TYPE ST_AxisError:
STRUCT
//PLCopen function block errors
    nPowerErrorID: UDINT; //Error ID MC_Power function block
    nMoveAbsoluteErrorID: UDINT; //Error ID for MC_MoveAbsolute function block
    nMoveRelativeErrorID: UDINT; //Error ID for MC_MoveRelative function block
    nMoveVelocityErrorID: UDINT; //Error ID for MC_MoveVelocity function block
    nMoveModuloErrorID: UDINT; //Error ID for MC_MoveModulo function block
    nHomeErrorID: UDINT; //Error ID for MC_Home function block
    nHaltErrorID: UDINT; //Error ID for MC_Halt function block
    nResetErrorID: UDINT; //Error ID for MC_Reset function block
    nStopErrorID: UDINT;//Error ID for MC_Stop function block
    nGearInMultiMasterErrorID: UDINT; //Error ID for MC_GearInMultiMaster function block
    nGearOutErrorID: UDINT; //Error ID for MC_GearOut function block
    nWriteParameterErrorID: UDINT; //Error ID for writing parameters function block
    nReadParameterErrorID: UDINT; //Error ID for MC_ReadParameter function block
    nBacklashErrorID: UDINT; //Error ID for MC_BacklashCompensation function block
    nTempDisableErrorID: UDINT; //Error ID for mControl_TemperatureDisable method
    nCommandHandlerErrorID: UDINT; //Error ID for mControl_CommandHandler method
    nAirpadErrorID: UDINT; //Error ID for mControl_Airpad method
    nExternalBrakeErrorID: UDINT; //Error ID for mControl_ExternalBrake method
//Error from the NC
    nNCErrorID: UDINT; //Error ID from the NC Axis_Ref Axis Status
END_STRUCT
END_TYPE

(* stored: Version 1.1.0.1
   DUT ST_AxisError: Id {4d23f353-6484-09b3-1cf9-9d08ea568830} *)
